TEXTLIST TextList_Util_Userlist
  4 = 'Liste des utilisateurs' | FR: 'Liste des utilisateurs' | EN: 'User list'
  5 = 'Liste des groupes' | FR: 'Liste des groupes' | EN: 'Group list'
  1 = 'Create user' | FR: "Création d'un nouvel utilisateur" | EN: 'New user creation'
  2 = 'user info' | FR: "Informations sur l'utilisateur" | EN: 'User information'
  3 = 'choix groupe' | FR: 'Sélection du groupe' | EN: 'Group selection'
  0 = 'Modify user' | FR: "Modification d'un utilisateur" | EN: 'User modification'
   = ''
END_TEXTLIST

(* stored: Version 1.1.0.1, ProductVersion 3.1.4024.10
   TextList TextList_Util_Userlist: Id {8c1ac405-d2b5-444c-9e48-e1430bdf654a} *)
